// This function has been automatically generated from the project information.
{attribute 'signature_flag' := '1073741824'}
{attribute 'TcGenerated'}
{attribute 'no-analysis'}
FUNCTION F_GetTitle : WSTRING
VAR_INPUT
	
END_VAR

F_GetTitle := "Tc3_prx";

END_FUNCTION

(* stored: Version 1.1.0.1
   POU F_GetTitle: Id {b978736d-2f9c-425e-a9b4-bf52e7775988}, SpecialFunc None *)
